FUNCTION_BLOCK FB_PressureSensor EXTENDS StateMachineBase IMPLEMENTS I_PressureSensor
VAR_INPUT
    bIsSimulator : BOOL;
END_VAR
VAR_OUTPUT
END_VAR
VAR
    fInputSignal : LREAL; // 0-10v
    fBufferedSignal : LREAL; // 0-10v
END_VAR

METHOD getSignal : LREAL
VAR_INPUT
END_VAR
getSignal := 0;
END_METHOD

METHOD setSignal : BOOL
VAR_INPUT
    input : LREAL;
END_VAR
fInputSignal := input;
END_METHOD

END_FUNCTION_BLOCK

(* stored: Version 1.1.0.1, ProductVersion 3.1.4024.9
   POU FB_PressureSensor: Id {fc5cba41-ac72-4fd3-8065-3ed8fcbd0f20}, SpecialFunc None
   Method getSignal: Id {115ab3f5-275d-439f-ad08-838594ccf2d5}
   Method setSignal: Id {6f58a8cb-a92e-47f6-bbe4-f00f2e021398} *)
